(* PLC project robot6axis_ctrled, Dassault Systèmes ControlBuild 2024x *)
(* stored: creationDateTime 2023-10-04T11:04:01-01:00 *)

PROGRAM robot6axis_ctrled.robot6axis_ctrled
  VAR_INPUT
    armOrigin : ARRAY[1..3] OF REAL := [800.0, 400.0, 0.0];
    profileNr : DINT := 0;
  END_VAR
  VAR_INPUT
    HomeCmd : BOOL := false;
    MoveVelCmd : BOOL := false;
    MoveAbsCmd : BOOL := false;
    MoveVel1ManualCmd : BOOL := false;
    MoveVel2ManualCmd : BOOL := false;
    MoveAbs1ManualCmd : BOOL := false;
    MoveAbs2ManualCmd : BOOL := false;
    StopCmd : BOOL := false;
    MovePosition : REAL := 0.0;
    MoveSpeed : REAL := 100.0;
    MoveAcceleration : REAL := 100.0;
    MoveDeceleration : REAL := 100.0;
    offsetAxToMa : REAL := 0.0;
    gripSyringes : BOOL := false;
  END_VAR
  VAR_INPUT
    Auto : BOOL := false;
    Manu : BOOL := false;
    run : BOOL := false;
  END_VAR
  VAR_OUTPUT
    armExtrem : ARRAY[1..3] OF REAL := [3(0.0)];
    velX : REAL := 0.0;
    velY : REAL := 0.0;
    velZ : REAL := 0.0;
    armInStop : BOOL := false;
  END_VAR
  VAR_OUTPUT
    masterPosition : REAL := 0.0;
    ActualPositionAx : REAL := 0.0;
  END_VAR

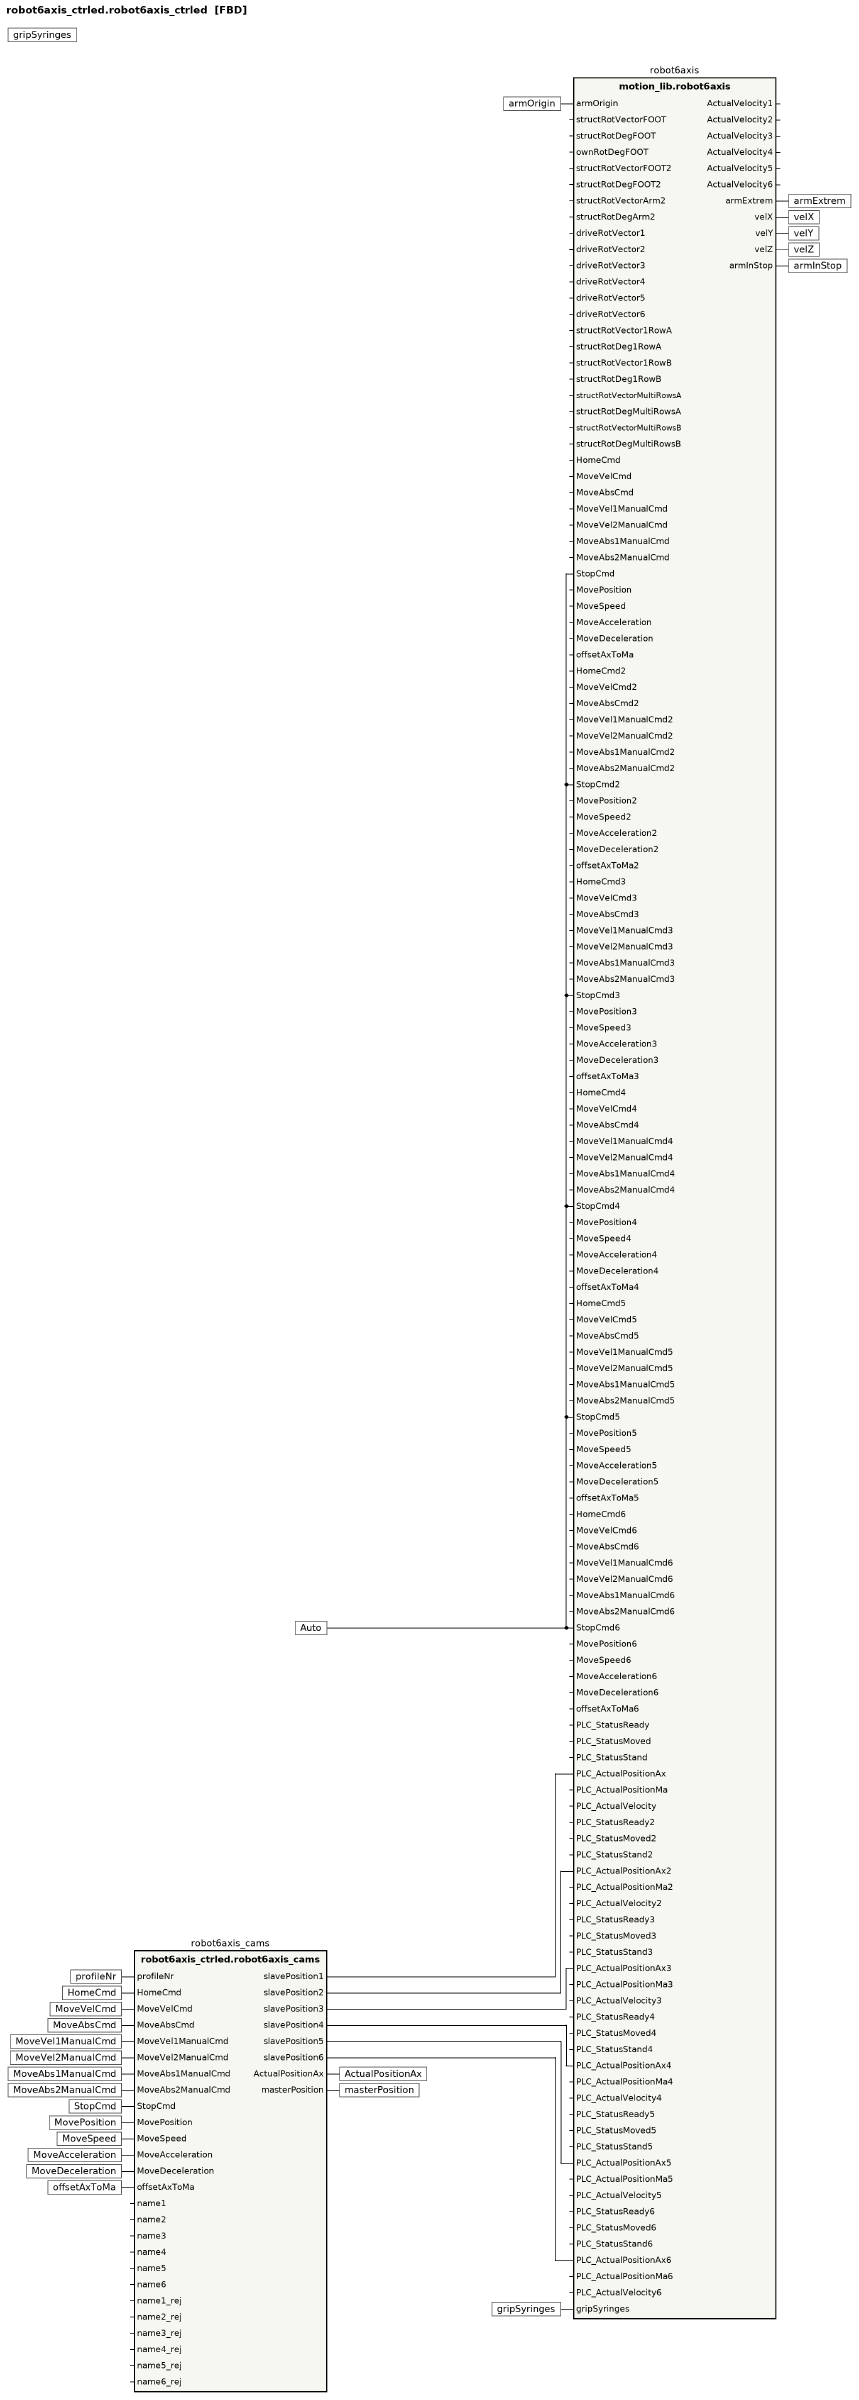
(* FBD diagram, written out as Structured Text *)
robot6axis_cams(profileNr := profileNr, HomeCmd := HomeCmd, MoveVelCmd := MoveVelCmd, MoveAbsCmd := MoveAbsCmd, MoveVel1ManualCmd := MoveVel1ManualCmd, MoveVel2ManualCmd := MoveVel2ManualCmd, MoveAbs1ManualCmd := MoveAbs1ManualCmd, MoveAbs2ManualCmd := MoveAbs2ManualCmd, StopCmd := StopCmd, MovePosition := MovePosition, MoveSpeed := MoveSpeed, MoveAcceleration := MoveAcceleration, MoveDeceleration := MoveDeceleration, offsetAxToMa := offsetAxToMa);
robot6axis(armOrigin := armOrigin, StopCmd := Auto, StopCmd2 := Auto, StopCmd3 := Auto, StopCmd4 := Auto, StopCmd5 := Auto, StopCmd6 := Auto, PLC_ActualPositionAx := robot6axis_cams.slavePosition1, PLC_ActualPositionAx2 := robot6axis_cams.slavePosition2, PLC_ActualPositionAx3 := robot6axis_cams.slavePosition3, PLC_ActualPositionAx4 := robot6axis_cams.slavePosition4, PLC_ActualPositionAx5 := robot6axis_cams.slavePosition5, PLC_ActualPositionAx6 := robot6axis_cams.slavePosition6, gripSyringes := gripSyringes);
armExtrem := robot6axis.armExtrem;
velX := robot6axis.velX;
velY := robot6axis.velY;
velZ := robot6axis.velZ;
armInStop := robot6axis.armInStop;
ActualPositionAx := robot6axis_cams.ActualPositionAx;
masterPosition := robot6axis_cams.masterPosition;
(* drawn but not wired to any output: gripSyringes *)
END_PROGRAM
